FUNCTION_BLOCK DigitalInspectorTests EXTENDS TcoCore._internals_TcoContext
VAR
	_sut : TcoInspectors.TcoDigitalInspector(THIS^);
	inspectedValue : BOOL;
	_result : TcoInspectors.eInspectorResult;
END_VAR

METHOD PROTECTED Main
CASE _testId OF
	eDigitalInspectorTests.Inspect:		
		THIS^.ProbeDoneWhen(_sut.Inspect(inspectedValue).Done);		
	eDigitalInspectorTests.GetResult:
		_result := _sut.Inspect(inspectedValue).Result;		
END_CASE
END_METHOD

END_FUNCTION_BLOCK

(* stored: Version 1.1.0.1, ProductVersion 3.1.4024.9
   POU DigitalInspectorTests: Id {8e88c5fb-6b37-0ee0-1dee-44bcdb0de8e4}, SpecialFunc None
   Method Main: Id {2386eb08-ae25-07fa-0ae2-18bdce87e272} *)
